TYPE Outfeed :
STRUCT
	roller : Roller;
	photo_sensor :ARRAY[0..1]OF FB_PhotoSensor;
END_STRUCT
END_TYPE

(* stored: Version 1.1.0.1, ProductVersion 3.1.4024.12
   DUT Outfeed: Id {a6d50419-4f72-4ed5-a78e-1edf9f2ec06a} *)
